// LS Electric XG5000 project: 과년67_3_4
// PLC NewPLC
// module base 0 slot 0: 입출력 모듈:XBC-DR20S (DC 24V 입력 12점, 릴레이 출력 8점)

PROGRAM NewProgram (task: 스캔 프로그램)

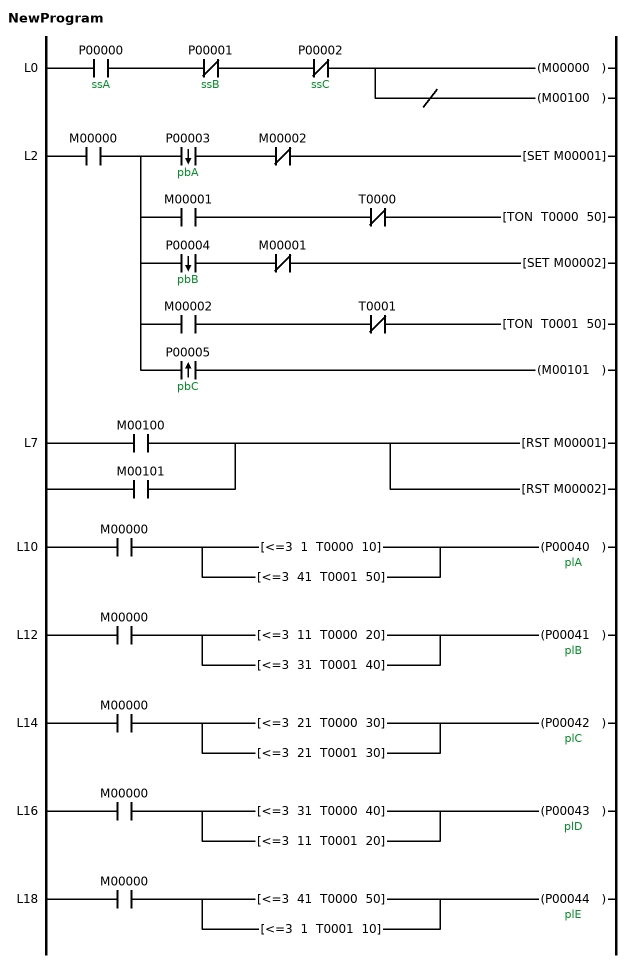
; L0
LOAD      P00000	// ssA
AND NOT   P00001	// ssB
AND NOT   P00002	// ssC
OUT       M00000
NOT
OUT       M00100
; L2
LOAD      M00000
MPUSH
ANDN      P00003	// pbA
AND NOT   M00002
SET       M00001
MLOAD
AND       M00001
AND NOT   T0000
TON       T0000 50
MLOAD
ANDN      P00004	// pbB
AND NOT   M00001
SET       M00002
MLOAD
AND       M00002
AND NOT   T0001
TON       T0001 50
MPOP
ANDP      P00005	// pbC
OUT       M00101
; L7
LOAD      M00100
OR        M00101
RST       M00001
RST       M00002
; L10
LOAD      M00000
LOAD<=3   1 T0000 10
OR<=3     41 T0001 50
AND LOAD
OUT       P00040	// plA
; L12
LOAD      M00000
LOAD<=3   11 T0000 20
OR<=3     31 T0001 40
AND LOAD
OUT       P00041	// plB
; L14
LOAD      M00000
LOAD<=3   21 T0000 30
OR<=3     21 T0001 30
AND LOAD
OUT       P00042	// plC
; L16
LOAD      M00000
LOAD<=3   31 T0000 40
OR<=3     11 T0001 20
AND LOAD
OUT       P00043	// plD
; L18
LOAD      M00000
LOAD<=3   41 T0000 50
OR<=3     1 T0001 10
AND LOAD
OUT       P00044	// plE